// TIA Portal V20 export
DATA_BLOCK "SBK8"   // DB292
// stored: MemoryReserve 100
   VAR
      "X1-1 LASER MARKING COVER UP/DOWN DETECT SENSOR" : Bool;
      "X2-1 WEIGHT NG MAGNETIC SAFETY DOOR SWITCH" : Bool;
      "X3-1 SPARE" : Bool;
      "X4-1 SPARE" : Bool;
      "X1-2 SPARE" : Bool;
      "X2-2 WEIGHT NG MAGNETIC SAFETY DOOR SWITCH" : Bool;
      "X3-2 SPARE" : Bool;
      "X4-2 SPARE" : Bool;
   END_VAR
BEGIN
END_DATA_BLOCK
